FUNCTION_BLOCK FB_SewMovitracBFieldbusTest EXTENDS FB_TestSuite
VAR_INPUT
END_VAR
VAR_OUTPUT
END_VAR
VAR
END_VAR

StartDrive();
HaltDrive();
RunWithSetSpeed();
ReadWarning();

METHOD HaltDrive : BOOL
VAR
	sut: FB_SewMovitracBFieldbus;
	control : ST_SimpleRotaryTwoWayDriveControl;
	result : UINT := 2#0000_1111_0000_0000; // SEW: Big Endian, TwinCAT: Little Endian
END_VAR
TEST('Halt drive');

control.Enable := TRUE;
control.Lock := TRUE;

sut(
	PI1 := 0,
	PI2 := 0,
	PI3 := 0,
	Control := control);
	
AssertEquals(result, sut.PO1.nUINT, 'Drive does not halt');

TEST_FINISHED();
END_METHOD

METHOD ReadWarning : BOOL
VAR_INPUT
END_VAR
VAR
	sut: FB_SewMovitracBFieldbus;
	result : BOOL := TRUE; 
END_VAR
TEST('Read warning');

sut(
	PI1 := 2#0010_0010_0000_0000,
	PI2 := 0,
	PI3 := 0);
	
AssertEquals(result, sut.Status.Warning, 'Warning not correctly decoded.');

TEST_FINISHED();
END_METHOD

METHOD RunWithSetSpeed : BOOL
VAR_INPUT
END_VAR
VAR
	sut: FB_SewMovitracBFieldbus;
	control : ST_SimpleRotaryTwoWayDriveControl;
	result : UINT := 2#0000_0110_0000_0000; // SEW: Big Endian, TwinCAT: Little Endian 
	resultSpeed : UINT := HOST_TO_BE16(80);
END_VAR
TEST('Run with set speed');

control.Direction := E_Direction.Right_Forward_Up;
control.Enable := TRUE;
control.Run := TRUE;
control.Speed := 80;

sut(
	PI1 := 0,
	PI2 := 0,
	PI3 := 0, 
	Control := control);

AssertEquals(result, sut.PO1.nUINT, 'Drive does not run with set speed');
AssertEquals(resultSpeed, sut.PO2, 'Drive does not run with set speed');

TEST_FINISHED();
END_METHOD

METHOD StartDrive : BOOL
VAR
	sut: FB_SewMovitracBFieldbus;
	control : ST_SimpleRotaryTwoWayDriveControl;
	result : UINT := 2#0000_0110_0000_0000; // SEW: Big Endian, TwinCAT: Little Endian
END_VAR
TEST('Start drive');

control.Direction := E_Direction.Right_Forward_Up;
control.Enable := TRUE;
control.Run := TRUE;

sut(
	PI1 := 0,
	PI2 := 0,
	PI3 := 0,
	Control := control);
	
AssertEquals(result, sut.PO1.nUINT, 'Drive does not start');

TEST_FINISHED();
END_METHOD

END_FUNCTION_BLOCK

(* stored: Version 1.1.0.1, ProductVersion 3.1.4024.11
   POU FB_SewMovitracBFieldbusTest: Id {7bd8768f-1d83-4ed6-b68c-1803c627cd42}, SpecialFunc None
   Method HaltDrive: Id {1ae30293-fd52-4ea7-acbb-81956053393c}
   Method ReadWarning: Id {8e6c3be0-6ec9-42a6-a036-e1aaf21a8f48}
   Method RunWithSetSpeed: Id {967c6481-fbe4-4d33-99ef-e48f83a7e2de}
   Method StartDrive: Id {d3226732-84b5-46a5-80e4-6e0ce4e1734b} *)
